{attribute 'qualified_only'} var_config MAIN.fbMotor.bEnable at %QX0.0:bool; MAIN.fbMotor.nSpeed at %QW2:int; end_var

(* stored: Version 1.1.0.1, ProductVersion 3.1.4024.16
   GVL GVL_Syntax_Config: Id {c1d2e3f4-a5b6-4c7d-8e9f-0a1b2c3d4e5f} *)
